SUBAPPLICATION Uebung_001f (* DigitalInput_I1 negiert mit INIT auf DigitalOutput_Q1 *)
  (* Standard: 61499-2; Description: Copyright (c) 2023 Meisterschulen am Ostbahnhof This program and the accompanying materials are made available under the terms of the Eclipse Public License 2.0 which is available at https://www.eclipse.org/legal/epl-2.0/ SPDX-License-Identifier: EPL-2.0 *)
  (* Version 1.0, 2023-10-23, Franz Höpfinger, Meisterschulen am Ostbahnhof, initial API and implementation and/or initial documentation *)
  PACKAGE Uebungen;
  IMPORT logiBUS::io::DI::logiBUS_DI::Input_I1;
  IMPORT logiBUS::io::DQ::logiBUS_DO::Output_Q1;
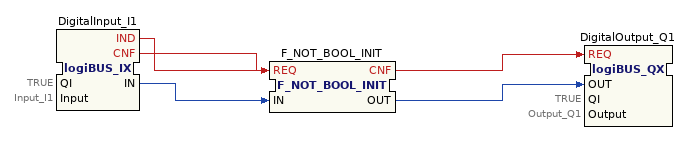
  (* obwohl I1 nicht abgefragt wird beim BOOT, wird AX_NOT hier TRUE ausgeben. *)
  FBS
    DigitalOutput_Q1 : logiBUS::io::DQ::logiBUS_QX(QI := TRUE, Output := Output_Q1);
    DigitalInput_I1 : logiBUS::io::DI::logiBUS_IX(QI := TRUE, Input := Input_I1);
    F_NOT_BOOL_INIT : iec61131::booleanOperators::F_NOT_BOOL_INIT;
  END_FBS
  EVENT_CONNECTIONS
    DigitalInput_I1.IND TO F_NOT_BOOL_INIT.REQ;
    DigitalInput_I1.CNF TO F_NOT_BOOL_INIT.REQ;
    F_NOT_BOOL_INIT.CNF TO DigitalOutput_Q1.REQ;
  END_CONNECTIONS
  DATA_CONNECTIONS
    DigitalInput_I1.IN TO F_NOT_BOOL_INIT.IN;
    F_NOT_BOOL_INIT.OUT TO DigitalOutput_Q1.OUT;
  END_CONNECTIONS
END_SUBAPPLICATION
